# B&R Automation Studio project GithubExample
Automation Studio 4.1.10.69 SP; Default project

## Configuration Simulation

CPU , AutomationRuntime L4.10

### Hardware
```
PC_any : PC_any v1.0.3.0 (OrderNumber=PC)
```


Listed in the project but not available here: Logical/Libraries
